// TIA Portal V17 export
// export: Created 2023-04-11T09:34:01.4736729Z, ExportSetting WithDefaults, DisplayName Totally Integrated Automation Portal, DisplayVersion V17 Update 3, DisplayName TIA Portal Openness, DisplayVersion V17 Update 3, DisplayName TIA Portal Version Control Interface, DisplayVersion V17, DisplayName SINAMICS Startdrive Advanced, DisplayVersion V17 Update2, DisplayName SINAMICS Startdrive G130, G150, S120, S150, SINAMICS MV, S210, DisplayVersion V17 Update2, DisplayName SINAMICS Startdrive G110M, G120, G120C, G120D, G120P, G115D, DisplayVersion V17 Update2, DisplayName STEP 7 Professional, DisplayVersion V17 Update 3, DisplayName STEP 7 Safety, DisplayVersion V17, DisplayName WinCC UA Professional, DisplayVersion V17 Update 3
FUNCTION_BLOCK "FB_iTacSettingLog"   // FB68, LAD
{ S7_Optimized_Access := 'FALSE' }
VERSION : 0.1
// stored: AutoNumber true, IsIECCheckEnabled false, SetENOAutomatically false, UDAEnableTagReadback false
   VAR_INPUT
      ID : UInt;
      reset : Bool;
      iTacConnectionEst : Bool;
      actualLoggedLevel : Int;
      dataDeliminer : String;
      errorText : String;
      errorSignalization : Bool;
      timeout_value : Time;
   END_VAR
   VAR_OUTPUT
      pass : Bool;
      fail : Bool;
      exception : Bool;
      testMap : String;
      timeout_err : Bool;
      retval : UInt;
   END_VAR
   VAR_IN_OUT
      data : Variant;
      dataRecieved : "t_LString";
      dataToSendOut : "t_LString";
      recipeControl : "t_recipeEKSLog";
      rettext_o : String;
   END_VAR
   VAR DB_SPECIFIC
      trig : Bool;
      sendingActive : Bool;
      sendedWaitForResp : Bool;
      freeForSend : Bool;
      changeEvent : Array[0..#numOfElem] of Bool;
      requestBuffer : Array[0..#numOfElem] of Bool;
      edge : Array[0..0] of Bool;
      Timeout { S7_SetPoint := 'True'} : TON_TIME;
   END_VAR
   VAR
      iPA_iTac_timeout { S7_SetPoint := 'True'} : Program_Alarm;
      iPA_iTac_fail { S7_SetPoint := 'True'} : Program_Alarm;
   END_VAR
   VAR DB_SPECIFIC
      toutErr : Bool;
      retValStr : String;
      number : UDInt;
      pos : DInt;
      ret_val : Int;
      byteArr : Array[0..999] of Byte;
      dataToSendPrepareBuffer { S7_SetPoint := 'True'} : "t_LString";
      dataToSendBuffer { S7_SetPoint := 'True'} : "t_LString";
      actNumOfChanges : Int;
      lastRecipeSendMessage : Int;
      recipeLoadIndex : Int;
      recipeLoaded : Bool;
      monitor1 : Int;
   END_VAR
   VAR_TEMP
      id_x : UInt;
      id_x1 : Bool;
      id_x9 : Bool;
      fail_local : Bool;
      pass_local : Bool;
      auxStr : String;
      ID_recieved : UInt;
      sendPLS : Bool;
      i : Int;
      settingsLogging : Array[0..#numOfElem] of "tSwitchOnOff_log";   // max 20 values
      elemCount : Int;
      changeFlag : SInt;
      failTac : Bool;
      ID_lstring : "t_LString";
      buffDi : DWord;
      changeEventErase : Array[0..#numOfElem] of Bool;
   END_VAR
   VAR CONSTANT
      numOfElem : Int := 31;
      sizeOfElem : Int := 20;
   END_VAR
   VAR_TEMP   // added for the SCL form of the ladder/FBD networks
      _w1 : Bool;
      _w2 : Bool;
      _w3 : Bool;
   END_VAR
BEGIN

REGION Network 1: reset / init
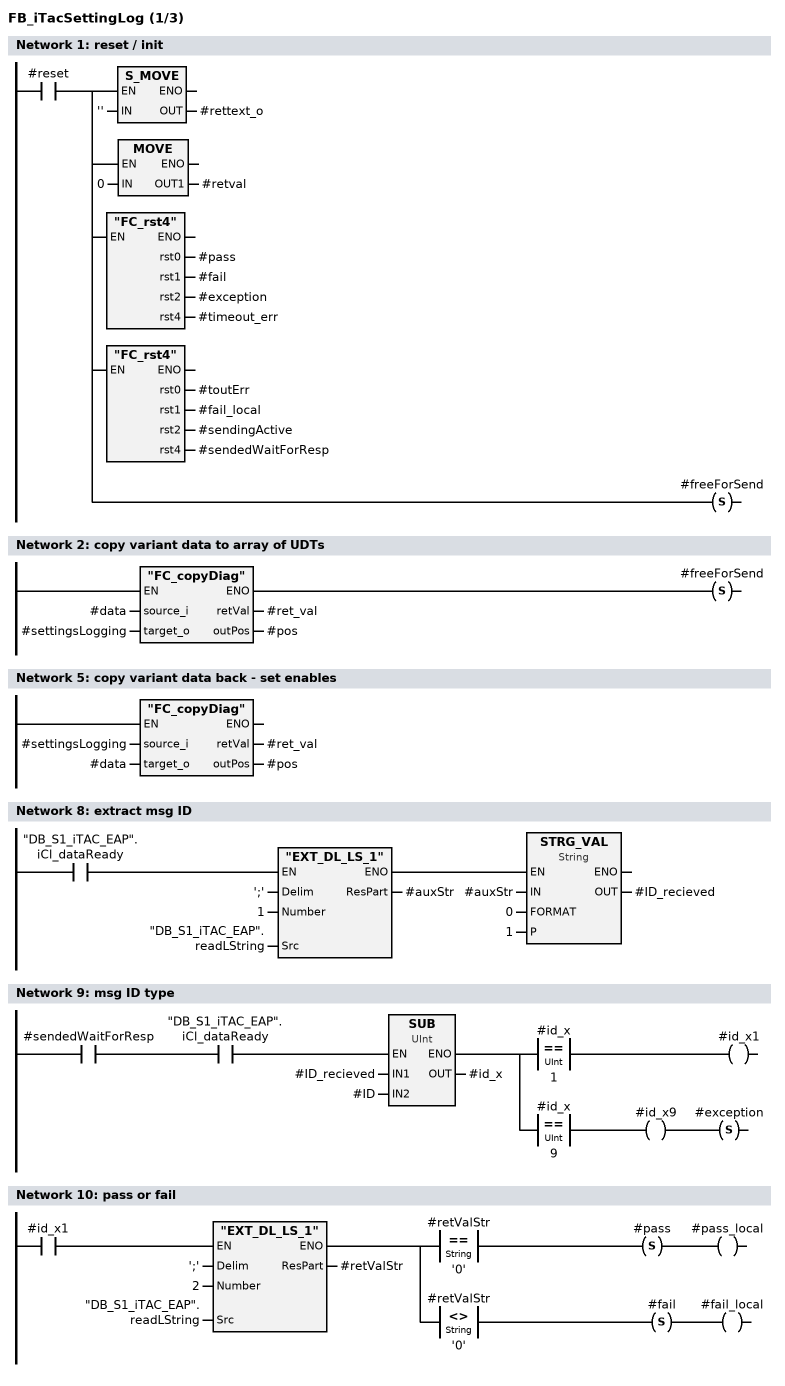
   RUNG wire#powerrail
      Contact( #reset )
      wire#w1
      S_Move(in := '', out => #rettext_o)
   END_RUNG
   RUNG wire#w1
      Move(in := 0, out1 => #retval)
   END_RUNG
   RUNG wire#w1
      "FC_rst4"(rst0 => #pass, rst1 => #fail, rst2 => #exception, rst4 => #timeout_err)
   END_RUNG
   RUNG wire#w1
      "FC_rst4"(rst0 => #toutErr, rst1 => #fail_local, rst2 => #sendingActive, rst4 => #sendedWaitForResp)
   END_RUNG
   RUNG wire#w1
      S_Coil( #freeForSend )
   END_RUNG
   // the same network as SCL:
   IF #reset THEN
       #rettext_o := '';
       #retval := 0;
       "FC_rst4"(rst0 => #pass, rst1 => #fail, rst2 => #exception, rst4 => #timeout_err);
       "FC_rst4"(rst0 => #toutErr, rst1 => #fail_local, rst2 => #sendingActive, rst4 => #sendedWaitForResp);
       #freeForSend := TRUE;
   END_IF;
END_REGION

REGION Network 2: copy variant data to array of UDTs
   RUNG wire#powerrail
      "FC_copyDiag"(source_i := #data, target_o := #settingsLogging, retVal => #ret_val, outPos => #pos)
      S_Coil( #freeForSend )
   END_RUNG
   // the same network as SCL:
   "FC_copyDiag"(source_i := #data,
                 target_o := #settingsLogging,
                 retVal => #ret_val,
                 outPos => #pos,
                 ENO => #_w1);
   IF #_w1 THEN #freeForSend := TRUE; END_IF;
END_REGION

REGION Network 3 (SCL)
   #elemCount := DINT_TO_INT(#pos / #sizeOfElem);
END_REGION

REGION Network 4 (SCL)
   FOR #i := 0 TO #elemCount - 1 DO
       #settingsLogging[#i].enable := #settingsLogging[#i].secLevel <= #actualLoggedLevel;
   END_FOR;
END_REGION

REGION Network 5: copy variant data back - set enables
   RUNG wire#powerrail
      "FC_copyDiag"(source_i := #settingsLogging, target_o := #data, retVal => #ret_val, outPos => #pos)
   END_RUNG
   // the same network as SCL:
   "FC_copyDiag"(source_i := #settingsLogging, target_o := #data, retVal => #ret_val, outPos => #pos);
END_REGION

REGION Network 7 (SCL): check changed value
   // Find number of elements

   #changeFlag := 0; // for cycle time optimalize
   #changeEvent := #changeEventErase;

   // Find request changed of elements
   FOR #i := 0 TO (#elemCount - 1) DO
       #changeEvent[#i] := #requestBuffer[#i] <> #settingsLogging[#i].actState;

       IF #changeEvent[#i] THEN
           #sendingActive := true;
           #changeFlag := #changeFlag + 1;
       END_IF;

       #requestBuffer[#i] := (#settingsLogging[#i].actState);
   END_FOR;

   #monitor1 := #monitor1 + #changeFlag;
   // Prepare send string
   IF #changeFlag > 0 THEN
       // copy ID
       #actNumOfChanges := #actNumOfChanges + #changeFlag;
       IF NOT #sendingActive THEN
           "CLEAR_LS_1"(IN := #dataToSendPrepareBuffer);
       END_IF;

       // Header is added before send (count num. of elements)
   (*    IF NOT #sendingActive THEN
           "TO_LS"(IN := #ID, OUT := #dataToSendPrepareBuffer);

           "CONCAT_LS"(IN1 := #dataToSendPrepareBuffer,
                       IN2 := #dataDeliminer,
                       OUT := #dataToSendPrepareBuffer);

           "CONCAT_LS"(IN1 := #dataToSendPrepareBuffer,
                       IN2 := #changeFlag,
                       OUT := #dataToSendPrepareBuffer);
       ELSE


       END_IF;
       *)

       "CONCAT_LS_1"(IN1 := #dataToSendPrepareBuffer,
                   IN2 := #changeFlag,
                   OUT := #dataToSendPrepareBuffer);

       FOR #i := 0 TO (#elemCount - 1) DO
           IF (#changeEvent[#i] = true) THEN

               "CONCAT_LS_1"(IN1 := #dataToSendPrepareBuffer,
                           IN2 := #dataDeliminer,
                           OUT := #dataToSendPrepareBuffer);

               "CONCAT_LS_S_1"(IN1 := #dataToSendPrepareBuffer,
                             IN2 := #settingsLogging[#i].iTacText,
                             OUT := #dataToSendPrepareBuffer);

               "CONCAT_LS_1"(IN1 := #dataToSendPrepareBuffer,
                           IN2 := #dataDeliminer,
                           OUT := #dataToSendPrepareBuffer);

               "CONCAT_LS_1"(IN1 := #dataToSendPrepareBuffer,
                           IN2 := #settingsLogging[#i].actState,
                           OUT := #dataToSendPrepareBuffer);

           END_IF;
       END_FOR;

   END_IF;
   (*
   IF #sendingActive AND #freeForSend THEN
       "TO_LS"(IN := #ID, OUT := #ID_lstring);

           "CONCAT_LS"(IN1 := #ID_lstring,
                       IN2 := #dataToSendPrepareBuffer,
                       OUT := #dataToSendPrepareBuffer);

           "CONCAT_LS"(IN1 := #dataToSendPrepareBuffer,
                       IN2 := #dataDeliminer,
                       OUT := #dataToSendPrepareBuffer);

           "CONCAT_LS"(IN1 := #dataToSendPrepareBuffer,
                       IN2 := #actNumOfChanges,
                       OUT := #dataToSendPrepareBuffer);
   END_IF; *)
   // Send to iTac vs. save to HMI
   // 

   IF #sendingActive AND #freeForSend THEN
       IF #iTacConnectionEst THEN
           #dataToSendOut := #dataToSendPrepareBuffer;
           #sendedWaitForResp := 1;
           #sendingActive := false;
           "CLEAR_LS_1"(#dataToSendPrepareBuffer);
       ELSE
           #recipeControl.dataOut := #dataToSendPrepareBuffer;
           "CLEAR_LS_1"(#dataToSendPrepareBuffer);
           #sendingActive := false;
           #recipeControl.index := #recipeControl.index + 1;
           #recipeControl.saveComand := true;
       END_IF;
   END_IF;
END_REGION

REGION Network 8: extract msg ID
   RUNG wire#powerrail
      Contact( "DB_S1_iTAC_EAP".iCl_dataReady )
      "EXT_DL_LS_1"(Delim := ';', Number := 1, Src := "DB_S1_iTAC_EAP".readLString, ResPart => #auxStr)
      { S7_Templates := "[src_type := String, dest_type := UInt]" } STRG_VAL(IN := #auxStr, FORMAT := 0, P := 1, OUT => #ID_recieved)
   END_RUNG
   // the same network as SCL:
   "EXT_DL_LS_1"(EN := "DB_S1_iTAC_EAP".iCl_dataReady,
                 Delim := ';',
                 Number := 1,
                 Src := "DB_S1_iTAC_EAP".readLString,
                 ResPart => #auxStr,
                 ENO => #_w1);
   IF #_w1 THEN STRG_VAL(IN := #auxStr, FORMAT := 0, P := 1, OUT => #ID_recieved); END_IF;
END_REGION

REGION Network 9: msg ID type
   RUNG wire#powerrail
      Contact( #sendedWaitForResp )
      Contact( "DB_S1_iTAC_EAP".iCl_dataReady )
      { S7_Templates := "SrcType := UInt" } Sub(in1 := #ID_recieved, in2 := #ID, out => #id_x)
      wire#w1
      { S7_Templates := "SrcType := UInt" } EQ_Contact(in1 := #id_x, in2 := 1)
      Coil( #id_x1 )
   END_RUNG
   RUNG wire#w1
      { S7_Templates := "SrcType := UInt" } EQ_Contact(in1 := #id_x, in2 := 9)
      Coil( #id_x9 )
      S_Coil( #exception )
   END_RUNG
   // the same network as SCL:
   #_w1 := #sendedWaitForResp AND "DB_S1_iTAC_EAP".iCl_dataReady;
   IF #_w1 THEN #id_x := #ID_recieved - #ID; END_IF;
   #id_x1 := #_w1 AND (#id_x = 1);
   #id_x9 := #_w1 AND (#id_x = 9);
   IF #id_x9 THEN #exception := TRUE; END_IF;
END_REGION

REGION Network 10: pass or fail
   RUNG wire#powerrail
      Contact( #id_x1 )
      "EXT_DL_LS_1"(Delim := ';', Number := 2, Src := "DB_S1_iTAC_EAP".readLString, ResPart => #retValStr)
      wire#w1
      { S7_Templates := "SrcType := String" } EQ_Contact(in1 := #retValStr, in2 := '0')
      S_Coil( #pass )
      Coil( #pass_local )
   END_RUNG
   RUNG wire#w1
      { S7_Templates := "SrcType := String" } NE_Contact(in1 := #retValStr, in2 := '0')
      S_Coil( #fail )
      Coil( #fail_local )
   END_RUNG
   // the same network as SCL:
   "EXT_DL_LS_1"(EN := #id_x1,
                 Delim := ';',
                 Number := 2,
                 Src := "DB_S1_iTAC_EAP".readLString,
                 ResPart => #retValStr,
                 ENO => #_w1);
   #_w2 := #_w1 AND (#retValStr = '0');
   IF #_w2 THEN #pass := TRUE; END_IF;
   #pass_local := #_w2;
   #_w3 := #_w1 AND (#retValStr <> '0');
   IF #_w3 THEN #fail := TRUE; END_IF;
   #fail_local := #_w3;
END_REGION

REGION Network 11: iTac pass
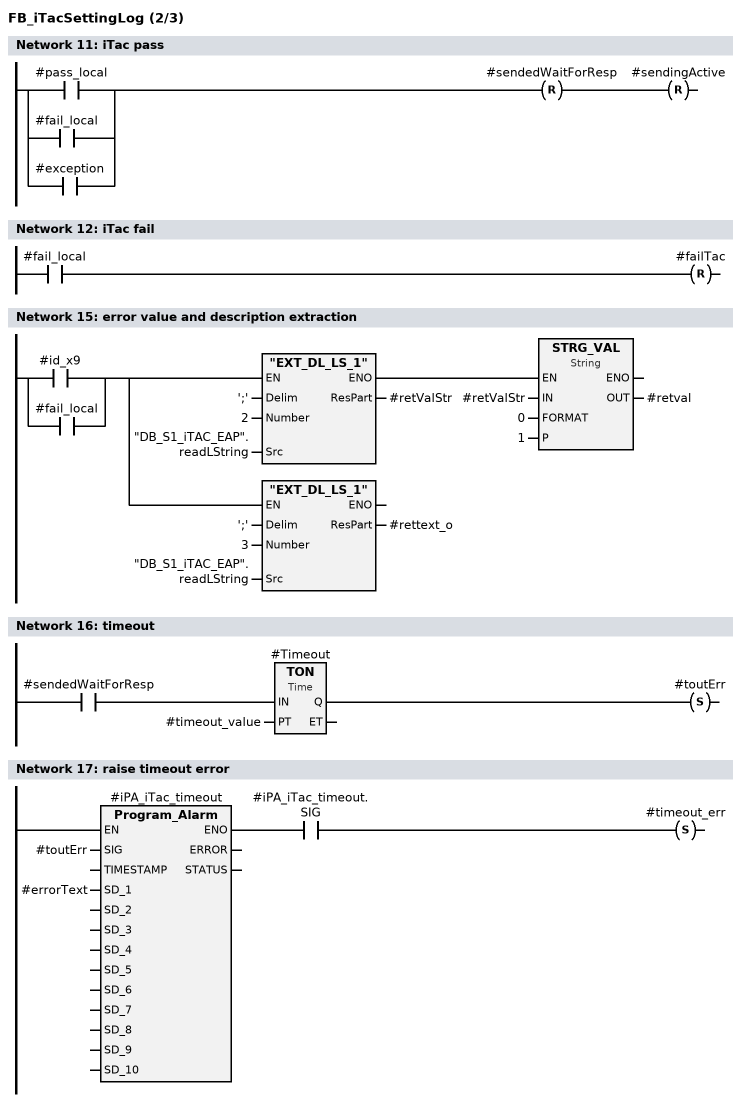
   RUNG wire#powerrail
      Contact( #pass_local )
      wire#w1
      R_Coil( #sendedWaitForResp )
      R_Coil( #sendingActive )
   END_RUNG
   RUNG wire#powerrail
      Contact( #fail_local )
   END_RUNG wire#w1
   RUNG wire#powerrail
      Contact( #exception )
   END_RUNG wire#w1
   // the same network as SCL:
   IF #pass_local OR #fail_local OR #exception THEN
       #sendedWaitForResp := FALSE;
       #sendingActive := FALSE;
   END_IF;
END_REGION

REGION Network 12: iTac fail
   RUNG wire#powerrail
      Contact( #fail_local )
      R_Coil( #failTac )
   END_RUNG
   // the same network as SCL:
   IF #fail_local THEN #failTac := FALSE; END_IF;
END_REGION

REGION Network 13 (SCL): pass - confirm ack signals
END_REGION

REGION Network 15: error value and description extraction
   RUNG wire#powerrail
      Contact( #id_x9 )
      wire#w1
      "EXT_DL_LS_1"(Delim := ';', Number := 2, Src := "DB_S1_iTAC_EAP".readLString, ResPart => #retValStr)
      { S7_Templates := "[src_type := String, dest_type := UInt]" } STRG_VAL(IN := #retValStr, FORMAT := 0, P := 1, OUT => #retval)
   END_RUNG
   RUNG wire#powerrail
      Contact( #fail_local )
   END_RUNG wire#w1
   RUNG wire#w1
      "EXT_DL_LS_1"(Delim := ';', Number := 3, Src := "DB_S1_iTAC_EAP".readLString, ResPart => #rettext_o)
   END_RUNG
   // the same network as SCL:
   "EXT_DL_LS_1"(EN := #id_x9 OR #fail_local,
                 Delim := ';',
                 Number := 2,
                 Src := "DB_S1_iTAC_EAP".readLString,
                 ResPart => #retValStr,
                 ENO => #_w1);
   IF #_w1 THEN STRG_VAL(IN := #retValStr, FORMAT := 0, P := 1, OUT => #retval); END_IF;
   IF #id_x9 OR #fail_local THEN
       "EXT_DL_LS_1"(Delim := ';', Number := 3, Src := "DB_S1_iTAC_EAP".readLString, ResPart => #rettext_o);
   END_IF;
END_REGION

REGION Network 16: timeout
   RUNG wire#powerrail
      Contact( #sendedWaitForResp )
      { S7_Templates := "time_type := Time" } #Timeout.TON(pt := #timeout_value, et =>)
      S_Coil( #toutErr )
   END_RUNG
   // the same network as SCL:
   #Timeout(IN := #sendedWaitForResp, PT := #timeout_value);   // TON
   IF #Timeout.Q THEN #toutErr := TRUE; END_IF;
END_REGION

REGION Network 17: raise timeout error
   RUNG wire#powerrail
      #iPA_iTac_timeout.Program_Alarm(SIG := #toutErr, TIMESTAMP :=, SD_1 := #errorText, SD_2 :=, SD_3 :=, SD_4 :=, SD_5 :=, SD_6 :=, SD_7 :=, SD_8 :=, SD_9 :=, SD_10 :=, Error =>, Status =>)
      Contact( #iPA_iTac_timeout.SIG )
      S_Coil( #timeout_err )
   END_RUNG
   // the same network as SCL:
   #iPA_iTac_timeout(SIG := #toutErr, SD_1 := #errorText, ENO => #_w1);   // Program_Alarm
   IF #_w1 AND #iPA_iTac_timeout.SIG THEN #timeout_err := TRUE; END_IF;
END_REGION

REGION Network 18: raise fail error
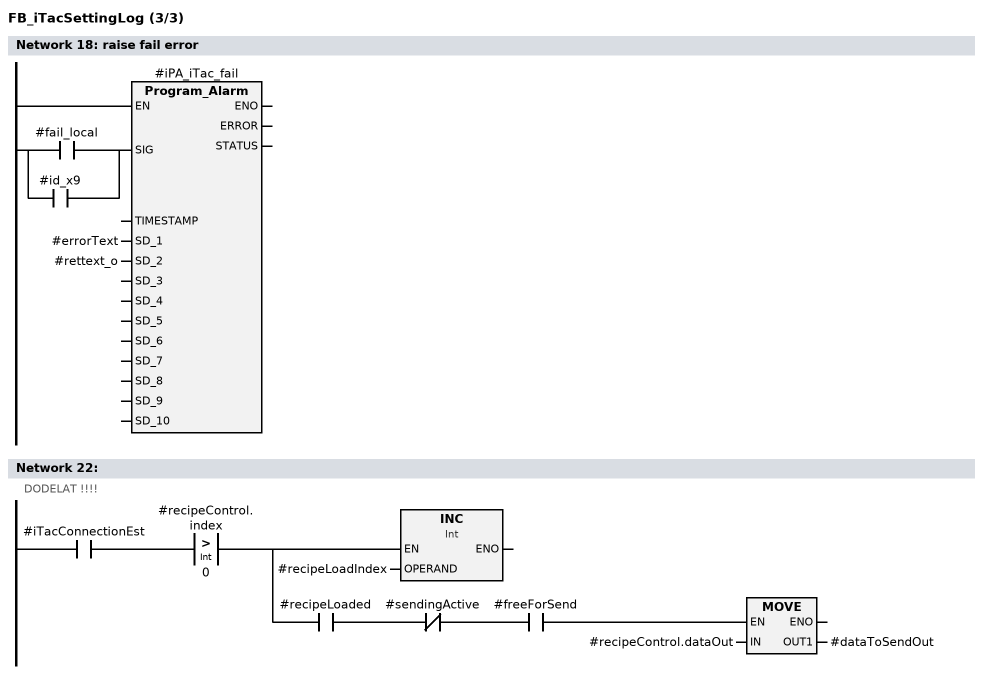
   RUNG wire#powerrail
      #iPA_iTac_fail.Program_Alarm(SIG := wire#w1, TIMESTAMP :=, SD_1 := #errorText, SD_2 := #rettext_o, SD_3 :=, SD_4 :=, SD_5 :=, SD_6 :=, SD_7 :=, SD_8 :=, SD_9 :=, SD_10 :=, Error =>, Status =>)
   END_RUNG
   RUNG wire#powerrail
      Contact( #fail_local )
   END_RUNG wire#w1
   RUNG wire#powerrail
      Contact( #id_x9 )
   END_RUNG wire#w1
   // the same network as SCL:
   #iPA_iTac_fail(SIG := #fail_local OR #id_x9, SD_1 := #errorText, SD_2 := #rettext_o);   // Program_Alarm
END_REGION

REGION Network 20 (SCL): prepareTestMap - string
   #testMap := '';
   (* GATHER(IN:=#requestBuffer,
          OUT=>#buffDi); *)
   #testMap := DINT_TO_STRING(IN := DWORD_TO_DINT(#buffDi));
   #testMap := DELETE(IN:=#testMap, L:=1, P:=1);
END_REGION

REGION Network 22
   // DODELAT !!!!
   RUNG wire#powerrail
      Contact( #iTacConnectionEst )
      { S7_Templates := "SrcType := Int" } GT_Contact(in1 := #recipeControl.index, in2 := 0)
      wire#w1
      { S7_Templates := "DestType := Int" } Inc( #recipeLoadIndex )
   END_RUNG
   RUNG wire#w1
      Contact( #recipeLoaded )
      I_Contact( #sendingActive )
      Contact( #freeForSend )
      Move(in := #recipeControl.dataOut, out1 => #dataToSendOut)
   END_RUNG
   // the same network as SCL:
   #_w1 := #iTacConnectionEst AND (#recipeControl.index > 0);
   IF #_w1 THEN #recipeLoadIndex := #recipeLoadIndex + 1; END_IF;
   IF #_w1 AND #recipeLoaded AND NOT #sendingActive AND #freeForSend THEN
       #dataToSendOut := #recipeControl.dataOut;
   END_IF;
END_REGION
END_FUNCTION_BLOCK
